(* IEC 61131-3 sources: axcoderepos/src, 3 files *)

(* ---- conveyor.st ---- *)
// using nmTankControl;
NAMESPACE Siemens.DemoMachine

    CLASS PUBLIC cConveyor
        VAR PUBLIC
            motor: IMotor;
            startSop: REF_TO BOOL;
        END_VAR

        VAR PRIVATE
            bb: BOOL ;
        END_VAR

        METHOD PUBLIC ConveyorControl

           IF startSop^ THEN
                motor.Run();
           ELSE
                motor.Stop();
            END_IF;
        END_METHOD
    END_CLASS

    INTERFACE IMotor
        METHOD Stop END_METHOD
        METHOD Run END_METHOD
    END_INTERFACE
    CLASS cMotor IMPLEMENTS IMotor
        VAR PUBLIC
            outRun: REF_TO BOOL;
        END_VAR
        METHOD PUBLIC Run
            outRun^ := TRUE;
        END_METHOD
        METHOD PUBLIC Stop
            outRun^ := FALSE;
        END_METHOD
        // METHOD PUBLIC MotorControl

        // END_METHOD
    END_CLASS
    CLASS cDriveMotor IMPLEMENTS IMotor
        VAR PUBLIC
            outSpeed: REF_TO REAL;
            outRun: REF_TO BOOL;
        END_VAR
        METHOD PUBLIC SetSpeed
            VAR_INPUT
                inSpeed: REAL;

            END_VAR

            IF inSpeed > 0.0 AND inSpeed < 60.0 THEN
                outSpeed^ := inSpeed;
            END_IF;
        END_METHOD
        METHOD PUBLIC Run
            outRun^ := TRUE;
        END_METHOD
        METHOD PUBLIC Stop
            outRun^ := FALSE;
        END_METHOD

    END_CLASS

END_NAMESPACE

(* ---- ConveyorFB.st ---- *)
NAMESPACE Siemens.DemoMachine.ConveyorUnit
FUNCTION_BLOCK PUBLIC ConveyorMotor
    VAR_INPUT
        startStop: BOOL;
    END_VAR
    VAR_OUTPUT
        outRun: BOOL;

    END_VAR
    VAR
        conveyor: cConveyor;
        motor: cMotor;

    END_VAR
        conveyor.startSop := REF(startStop);
        motor.outRun := REF(outRun);
        conveyor.motor := motor;
        conveyor.ConveyorControl();

END_FUNCTION_BLOCK

FUNCTION_BLOCK PUBLIC ConveyorDrive
    VAR_INPUT
        startStop: BOOL;
        speedSetpoint: REAL;
    END_VAR
    VAR_OUTPUT
        outRun: BOOL;
        outSpeed: REAL;
    END_VAR
    VAR
        conveyor: cConveyor;
        motor: cDriveMotor;
    END_VAR
    VAR_TEMP
        myrefbool: REF_TO BOOL;
    END_VAR
    // Run/Stop control
        conveyor.motor := motor;
        conveyor.startSop := REF(startStop);
        motor.outRun := REF(outRun);
        conveyor.ConveyorControl();
     // set drive speed
        motor.outSpeed := REF(outSpeed);
        motor.SetSpeed(speedSetpoint);

    ;
    //

END_FUNCTION_BLOCK

FUNCTION MyTestFC
    // VAR_IN_OUT
    // inout1:bool;
    // END_VAR
     VAR_INPUT
        in1: BOOL;
    END_VAR
    VAR_TEMP
        // myrefbool:REF_TO BOOL;
        tmpBool: BOOL;

        END_VAR

    // myrefbool^:=in1;
    tmpBool := in1;
END_FUNCTION

TYPE
    Colors: (RED, GREEN, BLUE);
END_TYPE

END_NAMESPACE

(* ---- CONFIGURATION.st ---- *)
USING Siemens.DemoMachine.ConveyorUnit;
CONFIGURATION PLC_1
    TASK Main(Interval := T#100ms, Priority := 1);
    PROGRAM P1 WITH Main : MainProgram;
    VAR_GLOBAL
        instConveyorMotor:ConveyorMotor;
        instConveyorDrive:ConveyorDrive;
    END_VAR
END_CONFIGURATION

PROGRAM MainProgram
    VAR

    END_VAR
    ;//1st test
END_PROGRAM
